FUNCTION_BLOCK A2X2_2X_TO_4AX (* Composite FB for convert A2X2 to 4 AX *)
  (* Standard: 61499-2; Function: A2X2 has 2 channels (UP/DOWN), each bidirectional, so it takes 4 unidirectional AX to represent it: IND_UP/IND_DOWN carry what A2X2 receives (its EO_UP/EO_DOWN indication side), REQ_UP/REQ_DOWN carry what gets sent out through A2X2 (its EI_UP/EI_DOWN request side).; Description: Copyright (c) 2026 HR Agrartechnik GmbH This program and the accompanying materials are made available under the terms of the Eclipse Public License 2.0 which is available at https://www.eclipse.org/legal/epl-2.0/ SPDX-License-Identifier: EPL-2.0 *)
  (* Version 1.0, 2026-08-31, Franz Höpfinger, HR Agrartechnik GmbH, Initial Version *)
  PACKAGE adapter::conversion::bidirectional;
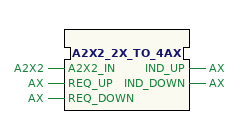
  SOCKETS
    A2X2_IN : adapter::types::bidirectional::A2X2; (* Adapter Input *)
    REQ_UP : adapter::types::unidirectional::AX; (* Request UP, received from outside, forwarded into A2X2_IN.EI_UP *)
    REQ_DOWN : adapter::types::unidirectional::AX; (* Request DOWN, received from outside, forwarded into A2X2_IN.EI_DOWN *)
  END_SOCKETS
  PLUGS
    IND_UP : adapter::types::unidirectional::AX; (* Indication UP, published outward from A2X2_IN.EO_UP *)
    IND_DOWN : adapter::types::unidirectional::AX; (* Indication DOWN, published outward from A2X2_IN.EO_DOWN *)
  END_PLUGS
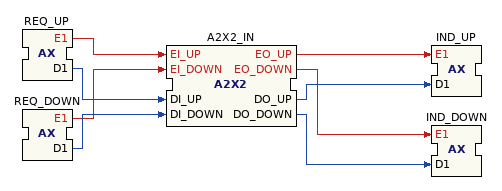
  EVENT_CONNECTIONS
    A2X2_IN.EO_UP TO IND_UP.E1;
    A2X2_IN.EO_DOWN TO IND_DOWN.E1;
    REQ_UP.E1 TO A2X2_IN.EI_UP;
    REQ_DOWN.E1 TO A2X2_IN.EI_DOWN;
  END_CONNECTIONS
  DATA_CONNECTIONS
    A2X2_IN.DO_UP TO IND_UP.D1;
    A2X2_IN.DO_DOWN TO IND_DOWN.D1;
    REQ_UP.D1 TO A2X2_IN.DI_UP;
    REQ_DOWN.D1 TO A2X2_IN.DI_DOWN;
  END_CONNECTIONS
END_FUNCTION_BLOCK
